Universal Robots PolyScope program: dummy.urp

Program dummy (installation=default directory=/programs createdIn=5.17.3 lastSavedIn=5.17.3 robotSerialNumber=20246801938)
Calibrated DH parameters: a=[-0.000071, -0.790281, -0.600694, 0.000061, -0.000039, 0]; d=[0.236272, 604.465945, 132.116513, -736.382239, 0.159268, 0.154005]; alpha=[1.570254, -0.000567, 0.000559, 1.571709, -1.56999, 0]; deltaTheta=[0, -0.409357, 7.293326, -0.600784, -0.000001, -0.000001]
InitVariablesNode
Robot Program (runOnlyOnce=true)
  SuppressedNode
    URCap MachineLogic for Universal Robots (MachineLogic for Universal Robots, Vention Inc.) dataModel(type=addMotor, numberAdded=0, speed_in_mm_per_min=600, acceleration_in_mm_per_s2=50.0, ActuatorPos=10.0, teachColor=BLUE, combo1=MachineMotion1, combo2=(1) Custom Actuator, combo3=Move Relative, combo6=In series, message=Move Rel., description=Moves the actuator away from its current position by a given distance., comboAddress=Address 1, comboActuator=Valve 1)
  SuppressedNode
    URCap MachineLogic for Universal Robots (MachineLogic for Universal Robots, Vention Inc.) dataModel(type=addMotor, numberAdded=0, ActuatorPos=800.0, speed_in_mm_per_min=4800.0, acceleration_in_mm_per_s2=20.0, teachColor=BLUE, combo1=MachineMotion1, combo2=(1) Custom Actuator, combo3=Move to Position, combo6=In series, message=Move to Position, description=Moves the actuator to a specified position from the home location., comboAddress=Address 1, comboActuator=Valve 1)
  SuppressedNode
    URCap MachineLogic for Universal Robots (MachineLogic for Universal Robots, Vention Inc.) dataModel(type=addMotor, numberAdded=0, ActuatorPos=0.0, acceleration_in_mm_per_s2=5.0, speed_in_mm_per_min=4800.0, teachColor=BLUE, combo1=MachineMotion1, combo2=(1) Custom Actuator, combo3=Move to Position, combo6=In series, message=Move to Position, description=Moves the actuator to a specified position from the home location., comboAddress=Address 1, comboActuator=Valve 1)
  SuppressedNode
    uh := [0,0,0]
  URCap WireTank Serial (WireTank Serial, WireTank, LLC) dataModel(QUERY=false, Command=[252,72,48], NODE_TITLE=Serial Bridge uH0, OUTPUT_ENTRY=Static, byte_array=true, Variable(key=OUTPUT_VARIABLE, variable=uh))
  URCap WireTank Serial (WireTank Serial, WireTank, LLC) dataModel(NODE_TITLE=Serial Bridge uh?, Command=[252,104,63], byte_array=true, QUERY=true, OUTPUT_ENTRY=Static, Variable(key=OUTPUT_VARIABLE, variable=uh))
  Popup Message (haltProgram=false inputType=Variable) variable=uh
  URCap WireTank Serial (WireTank Serial, WireTank, LLC) dataModel(byte_array=true, NODE_TITLE=Serial Bridge uH1, Command=[252,72,49], OUTPUT_ENTRY=Static, QUERY=false, Variable(key=OUTPUT_VARIABLE, variable=uh))
  URCap WireTank Serial (WireTank Serial, WireTank, LLC) dataModel(NODE_TITLE=Serial Bridge uh?, Command=[252,104,63], byte_array=true, QUERY=true, OUTPUT_ENTRY=Static, Variable(key=OUTPUT_VARIABLE, variable=uh))
  Popup Message (haltProgram=false inputType=Variable) variable=uh
